// TwinCAT 3 PLC project mobject_disposable
// Title: mobject-disposable
// Company: mobject
// Author: mobject dev team
// ProjectVersion: 1.0.0
// ProgramVersion: 3.1.4023.0
// project tree:
//   Disposable/ Disposable.TcPOU
//   Interfaces/ I_Disposable.TcIO

// ---- Interfaces/I_Disposable.TcIO
INTERFACE PUBLIC I_Disposable EXTENDS __System.IQueryInterface

METHOD PUBLIC Dispose
END_METHOD

END_INTERFACE

// ---- Disposable/Disposable.TcPOU
{attribute 'linkalways'} 
{attribute 'no_explicit_call' := 'This FB is a CLASS and must be accessed using methods or properties'}
{attribute 'enable_dynamic_creation'}
FUNCTION_BLOCK ABSTRACT Disposable IMPLEMENTS I_Disposable
VAR
END_VAR

METHOD PUBLIC Dispose
VAR
	pThis : POINTER TO Disposable;
END_VAR
pThis := THIS;
__DELETE(pThis);
END_METHOD

METHOD FB_exit : BOOL
VAR_INPUT
	bInCopyCode : BOOL; // if TRUE, the exit method is called for exiting an instance that is copied afterwards (online change).
END_VAR
// by default you would return if this is an in copy code, i.e. online change to this class
IF bInCopyCode THEN
	RETURN;
END_IF

// A word of warning. FB_exit does not NOT operate in the same way as a typical inherited method. If a child class does not implement FB_exit then it does not
// gain this one for itself. 
// The system will automatically call each FB_exit on each layer of inheritance one by one, starting with the child class and making it's way to the parent.
// Therefore code in here will only be triggered once the system reaches this layer of the object's deletion. The child class and all of it's variables
// will already have had FB_exit called by the time we reach this point!
END_METHOD

END_FUNCTION_BLOCK
